// Detects rising-edge errors
FUNCTION_BLOCK FB_ErrorTriggers
VAR_INPUT
    nLeakLocations : BYTE;
END_VAR
VAR_IN_OUT CONSTANT
    stErrors : ST_ErrorStates; // Errors that have been detected
END_VAR
VAR_OUTPUT
    stNewErrors : St_ErrorStates; // Rising-edge errors
END_VAR
VAR
    // R_TRIG function blocks for detecting new errors
    fbLeakTrig : R_TRIG;
    fbLeakOpticalTableAmphosOnTrig : R_TRIG;
    fbLeakOpticalTableNoLaserTrig : R_TRIG;
    fbLeakOpcpaCarbideOnTrig : R_TRIG;
    fbLeakUnderTableTrig : R_TRIG;
    fbLeakInsideRacksTrig : R_TRIG;
    fbAmphosBeamTrig : R_TRIG;
    fbOpcpaBeamTrig : R_TRIG;
    fbMPCBeamTrig : R_TRIG;
    fbDumpChillerTrig : R_TRIG;
    fbBaseplateChillerTrig : R_TRIG;

END_VAR

fbLeakTrig(
    CLK := nLeakLocations <> E_LeakLocation.NO_LEAK,
);
fbLeakOpticalTableAmphosOnTrig(
    CLK := stErrors.bLeakOpticalTableAmphosOn,
    Q => stNewErrors.bLeakOpticalTableAmphosOn
);
fbLeakOpticalTableNoLaserTrig(
    CLK := stErrors.bLeakOpticalTableNoLaser,
    Q => stNewErrors.bLeakOpticalTableNoLaser
);
fbLeakOpcpaCarbideOnTrig(
    CLK := stErrors.bLeakOpcpaCarbideOn,
    Q => stNewErrors.bLeakOpcpaCarbideOn
);
fbLeakUnderTableTrig(
    CLK := stErrors.bLeakUnderTable,
    Q => stNewErrors.bLeakUnderTable
);
fbLeakInsideRacksTrig(
    CLK := stErrors.bLeakInsideRacks,
    Q => stNewErrors.bLeakInsideRacks
);

fbAmphosBeamTrig(
    CLK := stErrors.bAmphosBeam,
    Q => stNewErrors.bAmphosBeam
);
fbOpcpaBeamTrig(
    CLK := stErrors.bOpcpaBeam,
    Q => stNewErrors.bOpcpaBeam
);

fbMPCBeamTrig(
    CLK := stErrors.bMPCBeam,
    Q => stNewErrors.bMPCBeam
);

fbDumpChillerTrig(
    CLK := stErrors.bDumpChiller,
    Q => stNewErrors.bDumpChiller
);
fbBaseplateChillerTrig(
    CLK := stErrors.bBaseplateChiller,
    Q => stNewErrors.bBaseplateChiller
);

// Returns whether a rising-edge leak error has occured
METHOD NewLeakError : BOOL
VAR_INPUT
END_VAR
NewLeakError := fbLeakTrig.Q OR fbLeakOpticalTableAmphosOnTrig.Q OR fbLeakOpticalTableNoLaserTrig.Q OR fbLeakOpcpaCarbideOnTrig.Q OR fbLeakUnderTableTrig.Q OR fbLeakInsideRacksTrig.Q;
END_METHOD

// Reset latched amphos errors
METHOD ResetAmphosTrigger
VAR_INPUT
END_VAR
fbAmphosBeamTrig(
    CLK := FALSE,
    Q => stNewErrors.bAmphosBeam
);
END_METHOD

METHOD ResetBaseplateChillerTrigger
VAR_INPUT
END_VAR
fbBaseplateChillerTrig(
    CLK := FALSE,
    Q => stNewErrors.bBaseplateChiller
);
END_METHOD

METHOD ResetDumpChillerTrigger
VAR_INPUT
END_VAR
fbDumpChillerTrig(
    CLK := FALSE,
    Q => stNewErrors.bDumpChiller
);
END_METHOD

// Reset latched leak errors
METHOD ResetLeakTriggers
VAR_INPUT
END_VAR
fbLeakOpticalTableAmphosOnTrig(
    CLK := FALSE,
    Q => stNewErrors.bLeakOpticalTableAmphosOn
);
fbLeakOpticalTableNoLaserTrig(
    CLK := FALSE,
    Q => stNewErrors.bLeakOpticalTableNoLaser
);
fbLeakOpcpaCarbideOnTrig(
    CLK := FALSE,
    Q => stNewErrors.bLeakOpcpaCarbideOn
);
fbLeakUnderTableTrig(
    CLK := FALSE,
    Q => stNewErrors.bLeakUnderTable
);
fbLeakInsideRacksTrig(
    CLK := FALSE,
    Q => stNewErrors.bLeakInsideRacks
);
END_METHOD

METHOD ResetMPCTrigger
VAR_INPUT
END_VAR
fbMPCBeamTrig(
    CLK := FALSE,
    Q => stNewErrors.bOpcpaBeam
);
END_METHOD

// Reset latched OPCPA errors
METHOD ResetOpcpaTrigger
VAR_INPUT
END_VAR
fbOpcpaBeamTrig(
    CLK := FALSE,
    Q => stNewErrors.bOpcpaBeam
);
END_METHOD

END_FUNCTION_BLOCK

(* stored: Version 1.1.0.1, ProductVersion 3.1.4022.18
   POU FB_ErrorTriggers: Id {03ec90dc-8712-481d-8a9d-9ad9d4cb604c}, SpecialFunc None
   Method NewLeakError: Id {ab5031be-34d4-41d7-8f1c-1e6706b02485}
   Method ResetAmphosTrigger: Id {ef779c79-51d0-48fb-aecc-a3d338593635}
   Method ResetBaseplateChillerTrigger: Id {5eeafa6d-3fc7-4559-abea-6ee754294cb1}
   Method ResetDumpChillerTrigger: Id {0e6a8265-2036-4d41-8243-aa7c141a7304}
   Method ResetLeakTriggers: Id {0cf9305f-aad5-4ef8-8c4c-82a427ee3c88}
   Method ResetMPCTrigger: Id {59b71cb5-2c00-4cd1-b0a7-f67ad33204d4}
   Method ResetOpcpaTrigger: Id {ac38f646-b9bb-4388-ba78-0da8d95694e7} *)
